Universal Robots PolyScope program: test to_string.urp

Program test to_string (installation=default directory=/programs createdIn=5.14.5 lastSavedIn=5.14.5 robotSerialNumber=20236801216)
Calibrated DH parameters: a=[-0.000021, -0.748897, -0.28186, -0.00004, -0.000055, 0]; d=[0.236225, -424.082933, -1564.66872, 1988.95162, 0.159094, 0.153873]; alpha=[1.570844, 0.001002, 0.000337, 1.571488, -1.569996, 0]; deltaTheta=[0, -0.516316, 5.626292, 1.173211, 0.000001, 0]
InitVariablesNode
Robot Program (runOnlyOnce=true)
  Script file /programs/test to_string file.script
    | x=12
    | list1=[x,2]
    | xs=str_cat("",x)
    | popup(xs)
  Popup Message (haltProgram=false inputType=Variable) variable(featureName=Point_1)
  Wait Sleep waitTime=50
